// TIA Portal V17 export
// export: Created 2025-01-08T13:55:35.415404Z, ExportSetting WithDefaults, DisplayName Totally Integrated Automation Portal, DisplayVersion V17, DisplayName TIA Portal Openness, DisplayVersion V17, DisplayName TIA Portal Version Control Interface, DisplayVersion V17, DisplayName SINAMICS Startdrive Advanced, DisplayVersion V17 Update2, DisplayName SINAMICS Startdrive G130, G150, S120, S150, SINAMICS MV, S210, DisplayVersion V17 Update2, DisplayName SINAMICS Startdrive G110M, G120, G120C, G120D, G120P, G115D, DisplayVersion V17 Update2, DisplayName STEP 7 Professional, DisplayVersion V17, DisplayName STEP 7 Safety, DisplayVersion V17, DisplayName WinCC Advanced, DisplayVersion V17
DATA_BLOCK "DB - Speed_2"   // DB89
{ S7_Optimized_Access := 'FALSE' }
VERSION : 0.1
// stored: AutoNumber true, DBAccessibleFromOPCUA true, DBAccessibleFromWebserver true, IsOnlyStoredInLoadMemory false, IsWriteProtectedInAS false
   VAR RETAIN
      SpeedSettings : "Speed_Change_Parameters";
   END_VAR
BEGIN
   SpeedSettings.LabelSpeed := 25;
   SpeedSettings.IndexWheelVelocity := 3000.0;
   SpeedSettings.IndexWheelAcceleration := 50000.0;
   SpeedSettings.IndexWheelDeceleration := 50000.0;
   SpeedSettings.IndexWheelJerk := 500000.0;
END_DATA_BLOCK
